FUNCTION_BLOCK BUBBLESIZEMETER (* Module that computes bubbles diameter on flotation froth *)
  (* Version 1.0, AN, SWDC RTSoft *)
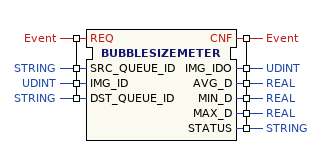
  EVENT_INPUT
    REQ WITH SRC_QUEUE_ID, IMG_ID, DST_QUEUE_ID;
  END_EVENT
  EVENT_OUTPUT
    CNF WITH IMG_IDO, AVG_D, MIN_D, MAX_D, STATUS;
  END_EVENT
  VAR_INPUT
    SRC_QUEUE_ID : STRING;
    IMG_ID : UDINT;
    DST_QUEUE_ID : STRING;
  END_VAR
  VAR_OUTPUT
    IMG_IDO : UDINT;
    AVG_D : REAL;
    MIN_D : REAL;
    MAX_D : REAL;
    STATUS : STRING;
  END_VAR
END_FUNCTION_BLOCK
